Fanuc KAREL source: kf00087.KL

-- PROVISIONAL review KL for V940-1; original PC SHA256 93176c6d914b6cea21e7fbd5ba14b25a224318d35956130a6f4bef354c8a5536
-- Incomplete behavior may be omitted. Consult companion uncertainty JSON. Do not deploy.
PROGRAM KF00087
%NOLOCKGROUP
BEGIN
  -- V9_ZERO_TABLE_METADATA_HINT layout=0002_ascii; no indexed target words; source/name/runtime held
  -- UNRESOLVED_PC offsets 5-28; opcodes 27,22,1C,31,4A
  -- UNRESOLVED_PC offsets 33-37; opcodes 7F
END KF00087
